GLOBALCONSTANTS AID_OM (* Output meter object attribute ids *)
  (* Standard: 61499-1; Description: Copyright (c) 2023 HR Agrartechnik GmbH This program and the accompanying materials are made available under the terms of the Eclipse Public License 2.0 which is available at https://www.eclipse.org/legal/epl-2.0/ SPDX-License-Identifier: EPL-2.0 *)
  (* Version 1.0, 2026-06-20, Franz Höpfinger, HR Agrartechnik GmbH *)
  PACKAGE isobus::UT::Q::const::AID;
  VAR_GLOBAL CONSTANT
    WIDTH : USINT := USINT#1; (* 1: AID_OM_WIDTH - Width in pixels. *)
    NEEDLE_COLOUR : USINT := USINT#2; (* 2: AID_OM_NEEDLE_COLOUR *)
    BORDER_COLOUR : USINT := USINT#3; (* 3: AID_OM_BORDER_COLOUR - Border colour index. *)
    ARC_THICK_COLOUR : USINT := USINT#4; (* 4: AID_OM_ARC_THICK_COLOUR *)
    OPTIONS : USINT := USINT#5; (* 5: AID_OM_OPTIONS - Bitmask: Bit 0=Draw Arc, Bit 1=Draw Border, Bit 2=Draw Ticks, Bit *)
    NUMB_TICKS : USINT := USINT#6; (* 6: AID_OM_NUMB_TICKS *)
    START_ANGLE : USINT := USINT#7; (* 7: AID_OM_START_ANGLE *)
    END_ANGLE : USINT := USINT#8; (* 8: AID_OM_END_ANGLE *)
    MIN_VALUE : USINT := USINT#9; (* 9: AID_OM_MIN_VALUE *)
    MAX_VALUE : USINT := USINT#10; (* 10: AID_OM_MAX_VALUE *)
    VARIABLE_REF : USINT := USINT#11; (* 11: AID_OM_VARIABLE_REF - Object ID of a Variable object. *)
    VALUE : USINT := USINT#12; (* 12: AID_OM_VALUE (read-only) - Current value. *)
  END_VAR
END_GLOBALCONSTANTS
